// SIMATIC S7-200 project (STEP 7-Micro/WIN), CPU 224 REL 01.22

SYMBOL_TABLE USR1
SAB3             I0.0     //  油泵电机启动
SAB4             I0.1     // 油泵电机停止
SAB5，6           I0.2     // 主轴正转
SAB7，8，9         I0.3     // 主轴停止
SAB10，11         I0.4     // 主轴反转
SAB12，13，14      I0.5     // 主轴正点动
SAB15，16，17      I0.6     // 主轴反点动
SP1，2，FR1        I0.7     // 油压正常
SL1              I1.0     // 回油泵启动
SL2              I1.1     // 回油泵制动
SQ3，SQ4          I1.2     // 主轴变档到位
SQ3，SQ5          I1.3     // 主轴变档到位
SQ3，SQ6          I1.4     // 主轴变档到位
SQ3，SQ7          I1.5     // 主轴变档到位
SP3              I2.0     // 过滤器堵塞
SP4              I2.1     // 过滤器堵塞
KAL1             I2.2     // 驱动器零速输出
KAL2             I2.3     // 驱动器正常输出
KAL3             I2.4     // 驱动器准备输出
SAB18            I2.5     // 套筒电机前进
SAB20            I2.6     // 套筒电机后退
SAB22            I2.7     // 尾座电机前进
SAB24            I3.0     // 尾座电机后退
SAB26            I3.1     // 左溜板箱油泵电机启动
SAB27            I3.2     // 左溜板箱油泵电机停止
SAB28            I3.3     // 左刀架油泵启动
SAB29            I3.4     // 移动停止
SAB30            I3.5     // 正转（前进）
SAB31            I3.6     // 反转（后退）
FR5              I3.7     // 溜板油泵保护
FR6              I4.0     // 刀架油泵保护
SQ8              I4.1     // 左刀架前进限位
SA3              I4.2     // 工作制选择-------给进
SA3，             I4.3     // 工作制选择-------快速
ZYZY             I4.5     // 左刀架1档---------左右
ZYQH             I4.4     // 左刀架1档---------前后
ZEZY             I4.7     // 左刀架2档---------左右
ZEQH             I4.6     // 左刀架2档---------前后
SQ9              I5.0     // 右刀架后退限位
SAB32            I5.1     // 右刀架溜板箱油泵电机启动
SAB33            I5.2     // 右刀架溜板箱油泵电机停止
SAB34            I5.3     // 右刀架油泵启动
SAB35            I5.4     // 右刀架移动停止
SAB36            I5.5     // 右刀架正转（前进）
SAB37            I5.6     // 右刀架反转（后退）
FR7              I5.7     // 右刀架溜板油泵保护
FR8              I6.0     // 刀架油泵保护
SQ10             I6.1     // 两刀架防相撞限位
SA6              I6.3     // 工作制选择----------给进
SA61             I6.2     // 工作制选择----------快速
YYZY             I6.6     // 右刀架1档---------左右
YYQH             I6.7     // 右刀架1档---------前后
YEZY             I6.4     // 右刀架2档---------左右
YEQH             I6.5     // 右刀架2档---------前进
KA0              I7.0     // 急停信号
SA5Y             I7.1     // 主轴变档--------1档
SA5E             I7.2     // 主轴变档--------2档
SA5S             I7.3     // 主轴变档--------3档
DYMKZBH          I7.4     // 驱动器信号
FR611            I7.5     // 驱动器过热信号
KSKZ611          I7.6     // 驱动器开始控制信号
SAB38，39         I7.7     // 主轴升速
SAB40，41         I8.0     // 主轴降速
SAB44，45         I8.7
KA1              Q0.0     // 油泵电机
KA2              Q0.1     // 辅助电源
KA3              Q0.2     // 油泵正常
KA4              Q0.3     // 主电机使能
KA5              Q0.4     // 主电机点动
KA6              Q0.5     // 主电机启动
KA7              Q0.6     // 油压报警
KA8              Q0.7     // 主轴变档电磁阀
KA9              Q1.0     // 主轴变档电磁阀
KA10             Q1.1     // 主轴变档电磁阀
KA11             Q2.0     // 主轴变档电磁阀
KA12             Q2.1     // 主轴1指示
KA13             Q2.2     // 主轴2指示
KA14             Q2.3     // 主轴3指示
HL12             Q2.4     // 过滤器清洗指示
HL13             Q2.5     // 过滤器清洗指示
KA15             Q2.6     // 套筒正转
KA16             Q2.7     // 套筒反转
KA17             Q3.0     // 尾座正转
KA18             Q3.1     // 尾座反转
HL14             Q3.2     // 快速移动指示
HL15             Q3.3     // 进给移动指示
HL16             Q3.4     // 左刀架-----横向移动1
HL17             Q3.5     // 左刀架-----横向移动2
HL18             Q3.6     // 左刀架-----纵向移动1
HL19             Q3.7     // 左刀架-----纵向移动2
KA19             Q4.0     // 左刀架变速传动-------1档
KA20             Q4.1     // 左刀架变速传动-------2档
KA21             Q4.2     // 左刀架变速纵向传动
KA22             Q4.3     // 左刀架变速横向传动
KA23             Q4.4     // 左刀架纵向制动
KA24             Q4.5     // 左刀架横向制动
KA25             Q4.6     // 左溜板油泵
KA26             Q4.7     // 左刀架油泵
KA27             Q5.0     // 回油泵（备用）
KA28             Q5.1
HL20             Q5.2     // 左刀架快速移动指示
HL21             Q5.3     // 左刀架给进移动指示
HL22             Q5.4     // 左刀架横向移动1
HL23             Q5.5     // 左刀架横向移动2
HL24             Q5.6     // 左刀架纵向移动1
HL25             Q5.7     // 左刀架纵向移动2
KA29             Q6.0     // 右刀架变速传动1档
KA30             Q6.1     // 右刀架变速传动2档
KA31             Q6.2     // 右刀架变速纵向传动
KA32             Q6.3     // 右刀架变速横向传动
KA33             Q6.4     // 右刀架变速纵向制动
KA34             Q6.5     // 右刀架变速横向制动
KA35             Q6.6     // 右溜板油泵
KA36             Q6.7     // 右刀架油泵
KA37             Q7.0     // 脉冲使能信号
KA38             Q7.1     // 控制使能信号
KA39             Q7.2     // 内部接触器控制
KA40             Q7.3     // 脉冲使能信号
KA41             Q7.4     // 控制使能信号
KA42             Q7.5     // 控制使能信号
KA43             Q7.6     // 选择电流控制方式
KA44             Q7.7     // 选择电流控制方式
KA45             Q8.1
KA46             Q8.2
KAJT             Q8.7
ZDJZZ            M1.0     // 左刀架正转标志位
ZDJFZ            M1.1     // 左刀架反转标志位
YDJZZ            M1.2     // 右刀架正转标志位
YDJFZ            M1.3     // 右刀架反转标志位
                 M5.2     // 主轴正转标志位
                 M5.3     // 主轴反转标志位
END_SYMBOL_TABLE

ORGANIZATION_BLOCK MAIN:OB1
TITLE=我设计了一个机床润滑系统的核心部件的程序。代码比较复杂，不知道具体实地应用如何，我写一下程序的实现目标以供参考。代码最后更新于2005年2月17号
// 实现目标：操作员通过主轴正转按钮、主轴反转按钮、主轴正点动按钮和主轴反点动按钮控制主轴方向，主电机启动信号驱动主轴连续旋转，主电机点动信号用于短暂调整。主轴模拟输出根据主轴升速按钮和主轴降速按钮调节转速。主轴1档选择开关、主轴2档选择开关和主轴3档选择开关分别触发主轴变档电磁阀1、主轴变档电磁阀2等，档位到位由主轴变档1到位传感器等确认，主轴1档指示灯等显示当前状态。
// 左刀架和右刀架可独立运行。左刀架正转按钮和左刀架反转按钮控制左刀架移动，右刀架正转按钮和右刀架反转按钮控制右刀架移动。左刀架给进模式开关和右刀架给进模式开关选择低速精确加工并调节左刀架模拟输出和右刀架模拟输出，左刀架快速模式开关和右刀架快速模式开关选择高速移动并调整相应输出。左刀架前进限位传感器和右刀架后退限位传感器防止超行程，左刀架防撞限位传感器检测两刀架距离。左刀架正转标志和右刀架反转标志的控制需注意避免相向移动导致碰撞，操作员应谨慎操作。
// 过滤器堵塞传感器1和过滤器堵塞传感器2检测到堵塞时，过滤器清洗指示灯1和过滤器清洗指示灯2亮起，提示维护。套筒电机前进按钮和套筒电机后退按钮分别驱动套筒正转信号和套筒反转信号。尾座电机前进按钮和尾座电机后退按钮分别驱动尾座正转信号和尾座反转信号。
// 紧急停止信号置位后，提示操作员机床处于停止状态。紧急停止按钮被按下时，紧急停止信号置位，操作员需手动复位油泵电机输出、主电机启动信号、套筒正转信号、尾座正转信号、主轴模拟输出、左刀架模拟输出和右刀架模拟输出，确保机床安全。
// 
BEGIN
Network 1
// 611驱动器准备
LD     SM0.0
CALL   SIEMENS611:SBR0
?000
Network 2
// 左刀架运行
LD     SM0.0
CALL   ZDJYX:SBR2
Network 3
// 右刀架运行
LD     SM0.0
CALL   YDJYX:SBR3
Network 4
// 主轴运行
LD     SM0.0
CALL   ZZYX:SBR1
Network 5
// 主轴模拟信号采样
LD     SM0.0
CALL   ZZMNXHCY:SBR4
Network 6
// 油泵电机启动
LD     SAB3:I0.0
O      KA1:Q0.0
AN     SAB4:I0.1
=      KA1:Q0.0
Network 7
// 过滤器清洗
LD     SP3:I2.0
=      HL12:Q2.4
Network 8
// 过滤器清洗
LD     SP4:I2.1
=      HL13:Q2.5
Network 9
// 套筒电机正转
LD     SAB18:I2.5
AN     SAB20:I2.6
=      KA15:Q2.6
Network 10
// 套筒电机反转
LD     SAB20:I2.6
AN     SAB18:I2.5
=      KA16:Q2.7
Network 11
// 尾座电机正转
LD     SAB22:I2.7
AN     SAB24:I3.0
=      KA17:Q3.0
Network 12
// 尾座电机反转
LD     SAB24:I3.0
AN     SAB22:I2.7
=      KA18:Q3.1
Network 13
// 回油泵工作
LD     SL1:I1.0
O      KA27:Q5.0
AN     SL2:I1.1
=      KA27:Q5.0
Network 14
LD     KA1:Q0.0
AN     SP1，2，FR1:I0.7
AN     T204
TON    T203, +20
Network 15
LD     T203
=      M12.0
TON    T204, +20
Network 16
// 报警
LDN    SP1，2，FR1:I0.7
LD     SAB5，6:I0.2
O      SAB10，11:I0.4
O      SAB12，13，14:I0.5
O      SAB15，16，17:I0.6
ALD
O      M12.0
=      KA7:Q0.6
Network 17
LDN    SAB44，45:I8.7
=      KAJT:Q8.7
END_ORGANIZATION_BLOCK

SUBROUTINE_BLOCK SIEMENS611:SBR0
TITLE=子例行程序注释
BEGIN
Network 1 // 网络标题
// 网络注释
LD     M7.0
AN     T108
=      KA39:Q7.2
TON    T250, +10
Network 2
LD     T250
AN     T107
=      KA37:Q7.0
TON    T101, +10
Network 3
LD     T101
AN     T106
=      KA38:Q7.1
TON    T102, +10
Network 4
LD     T102
AN     T105
LPS
TON    T103, +10
A      SA3:I4.2
=      KA43:Q7.6
LPP
A      SA6:I6.3
=      KA44:Q7.7
Network 5
LD     T103
AN     M7.1
=      KA40:Q7.3
Network 6
LD     M7.1
=      M0.0
TON    T105, +10
TON    T106, +20
TON    T107, +30
TON    T108, +40
Network 7
LD     SAB26:I3.1
O      SAB32:I5.1
LD     T109
NOT
A      M7.0
OLD
=      M7.0
Network 8
LD     M7.2
A      M7.3
LD     SAB26:I3.1
O      SAB32:I5.1
NOT
A      M7.1
OLD
=      M7.1
Network 9
LD     M7.1
=      M7.4
TON    T109, +45
Network 10
LD     SAB27:I3.2
LD     SAB26:I3.1
O      SAB32:I5.1
NOT
A      M7.2
OLD
=      M7.2
Network 11
LD     SAB33:I5.2
LD     SAB32:I5.1
O      SAB26:I3.1
NOT
A      M7.3
OLD
=      M7.3
END_SUBROUTINE_BLOCK

SUBROUTINE_BLOCK ZZYX:SBR1
TITLE=子例行程序注释
BEGIN
Network 1
// 辅助电源
LD     KA1:Q0.0
A      SP1，2，FR1:I0.7
=      KA2:Q0.1
TON    T37, +20
Network 2
// 停车信号
LD     T37
=      KA3:Q0.2
TON    T38, +20
Network 3
// 给启动信号
LD     T38
=      KA4:Q0.3
Network 4
// 正转标志位
LD     SAB5，6:I0.2
O      M5.2
LD     SAB7，8，9:I0.3
O      KA41:Q7.4
O      KA42:Q7.5
ALD
AN     SAB10，11:I0.4
AN     SAB15，16，17:I0.6
AN     SAB12，13，14:I0.5
A      KAL2:I2.3
=      M5.2
Network 5
// 反转标志位
LD     SAB10，11:I0.4
O      M5.3
LD     SAB7，8，9:I0.3
O      KA41:Q7.4
O      KA42:Q7.5
ALD
AN     SAB5，6:I0.2
AN     SAB15，16，17:I0.6
AN     SAB12，13，14:I0.5
A      KAL2:I2.3
=      M5.3
Network 6
// 主轴连动
LD     M5.2
O      M5.3
O      M24.0
O      M24.1
O      M25.0
O      M25.1
O      M25.2
A      SP1，2，FR1:I0.7
=      KA6:Q0.5
Network 7
LD     SAB12，13，14:I0.5
AN     SAB15，16，17:I0.6
=      M24.0
Network 8
LD     SAB15，16，17:I0.6
AN     SAB12，13，14:I0.5
=      M24.1
Network 9
LD     M24.0
O      M24.1
=      KA5:Q0.4
Network 10 // 网络标题
// 主轴变挡到位
LD     SQ3，SQ4:I1.2
=      M3.0
Network 11
// 主轴变挡到位
LD     SQ3，SQ5:I1.3
=      M3.1
Network 12
// 主轴变挡到位
LD     SQ3，SQ6:I1.4
=      M3.2
Network 13
// 主轴变挡到位
LD     SQ3，SQ7:I1.5
=      M3.3
Network 14
// 主轴1档
LD     SA5Y:I7.1
LDN    KAL1:I2.2
A      M3.4
OLD
AN     M3.6
AN     M4.0
=      M3.4
=      M3.5
Network 15
// 主轴1档指示灯
LD     M3.5
A      M3.1
A      M3.2
=      KA12:Q2.1
Network 16
// 主轴2档
LD     SA5E:I7.2
LDN    KAL1:I2.2
A      M3.6
OLD
AN     M3.4
AN     M4.0
=      M3.6
=      M3.7
Network 17
// 主轴2档指示灯
LD     M3.7
A      M3.0
A      M3.2
=      KA13:Q2.2
Network 18
// 主轴3档
LD     SA5S:I7.3
LDN    KAL1:I2.2
A      M4.0
OLD
AN     M3.4
AN     M3.6
=      M4.0
=      M4.1
Network 19
// 主轴3档指示灯
LD     M4.1
A      M3.1
A      M3.3
=      KA14:Q2.3
Network 20
// 电磁阀1
LD     M3.7
=      KA8:Q0.7
Network 21
// 电磁阀2
LD     M4.1
O      M3.5
=      KA9:Q1.0
Network 22
// 电磁阀3
LD     M3.5
O      M3.7
=      KA10:Q1.1
Network 23
// 电磁阀4
LD     M4.1
=      KA11:Q2.0
Network 24
// 1档换档脉动
LD     SA5Y:I7.1
LDN    M3.1
ON     M3.2
ALD
AN     T253
TON    T34, +800
Network 25
LDN    T34
TON    T253, +40
=      M25.0
Network 26
// 2档换档脉动
LD     SA5E:I7.2
LDN    M3.0
ON     M3.2
ALD
AN     T254
TON    T35, +200
Network 27
LD     T35
TON    T254, +40
=      M25.1
Network 28
// 3档换档脉动
LD     SA5S:I7.3
LDN    M3.1
ON     M3.3
ALD
AN     T255
TON    T36, +200
Network 29
LD     T36
TON    T255, +40
=      M25.2
END_SUBROUTINE_BLOCK

SUBROUTINE_BLOCK ZDJYX:SBR2
TITLE=子例行程序注释
BEGIN
Network 1
// 给定快速和给定速度范围
LD     SM0.0
LPS
A      SA3，:I4.3
LPS
A      M20.0
MOVW   +25000, AQW4
LPP
A      M20.1
MOVW   -25000, AQW4
LPP
A      SA3:I4.2
LPS
AW<=   AIW2, +32000
MOVW   AIW2, VW20
LPP
AW>=   AIW2, +32000
MOVW   +32000, VW20
Network 2
LD     SA3:I4.2
A      ZDJZZ:M1.0
AN     ZDJFZ:M1.1
MOVW   VW20, VW21
Network 3
// 选择速度范围
LD     SA3:I4.2
A      ZDJZZ:M1.0
AN     ZDJFZ:M1.1
AW<=   VW21, +32000
AW>=   VW21, +0
MOVW   VW21, AQW4
Network 4
// 改变方向
LD     SA3:I4.2
A      ZDJFZ:M1.1
AN     ZDJZZ:M1.0
MOVW   -1, VW200
*I     VW20, VW200
Network 5
LD     SA3:I4.2
A      ZDJFZ:M1.1
AN     ZDJZZ:M1.0
MOVW   VW200, VW201
Network 6
// 选择速度范围
LD     SA3:I4.2
A      ZDJFZ:M1.1
AN     ZDJZZ:M1.0
AW<=   VW201, +0
AW>=   VW201, -32000
MOVW   VW201, AQW4
Network 7
// 左溜板箱油泵电机
LD     SAB26:I3.1
O      KA25:Q4.6
AN     SAB27:I3.2
AN     FR5:I3.7
=      KA25:Q4.6
TON    T111, +3000
Network 8
// 左刀架油泵电机
LD     KA25:Q4.6
LD     SA3，:I4.3
LD     M20.0
O      M20.1
ALD
OLD
LDN    T111
O      M1.6
ALD
AN     FR6:I4.0
=      KA26:Q4.7
Network 9
// 左刀架油泵启动
LD     SAB28:I3.3
O      M1.6
AN     T112
=      M1.6
TON    T112, +3000
Network 10
// 左刀架工作方式选择
LD     KA25:Q4.6
LPS
AN     KAL1:I2.2
LD     SA3:I4.2
O      KA41:Q7.4
ALD
AN     HL14:Q3.2
=      HL15:Q3.3
LPP
A      SA3，:I4.3
AN     HL15:Q3.3
=      HL14:Q3.2
Network 11
// 左刀架1档左右
LD     KA25:Q4.6
LD     ZYZY:I4.5
O      KA41:Q7.4
ALD
AN     M2.0
AN     M2.1
AN     M2.2
=      HL16:Q3.4
=      M1.7
Network 12
// 左刀架1档前后
LD     KA25:Q4.6
LD     ZYQH:I4.4
O      KA41:Q7.4
ALD
AN     M1.7
AN     M2.1
AN     M2.2
=      HL18:Q3.6
=      M2.0
Network 13
// 左刀架2档左右
LD     KA25:Q4.6
LD     ZEZY:I4.7
O      KA41:Q7.4
ALD
AN     M1.7
AN     M2.0
AN     M2.2
=      HL17:Q3.5
=      M2.1
Network 14
// 左刀架2档前后
LD     KA25:Q4.6
LD     ZEQH:I4.6
O      KA41:Q7.4
ALD
AN     M1.7
AN     M2.0
AN     M2.1
=      HL19:Q3.7
=      M2.2
Network 15
// 左刀架电机正转
LD     SAB30:I3.5
O      ZDJZZ:M1.0
AN     SAB29:I3.4
A      SA3:I4.2
AN     ZDJFZ:M1.1
A      SQ8:I4.1
A      SP1，2，FR1:I0.7
AN     KAL1:I2.2
=      ZDJZZ:M1.0
Network 16
// 左刀架电机正点动
LD     SA3，:I4.3
AN     SA3:I4.2
A      SAB30:I3.5
AN     ZDJFZ:M1.1
=      M20.0
Network 17
// 左刀架电机反转
LD     SAB31:I3.6
O      ZDJFZ:M1.1
AN     SAB29:I3.4
A      SA3:I4.2
AN     ZDJZZ:M1.0
AN     SQ10:I6.1
A      SP1，2，FR1:I0.7
AN     KAL1:I2.2
=      ZDJFZ:M1.1
Network 18
// 左刀架电机反点动
LD     SA3，:I4.3
AN     SA3:I4.2
A      SAB31:I3.6
AN     ZDJZZ:M1.0
=      M20.1
Network 19
// 给定611启动信号
LD     ZDJZZ:M1.0
O      ZDJFZ:M1.1
AW>=   AIW2, +45
LD     M20.0
O      M20.1
OLD
=      KA41:Q7.4
Network 20
// 左刀架变速传动-------1档电磁阀
LD     M1.7
O      M2.0
A      SA3:I4.2
=      KA19:Q4.0
Network 21
// 给进状态下左刀架变速传动-------2档电磁阀标志位
LD     M2.1
O      M2.2
A      SA3:I4.2
=      M20.2
Network 22
// 快速状态下左刀架变速传动-------2档电磁阀标志位
LD     M2.1
O      M2.2
O      M1.7
O      M2.0
A      SA3，:I4.3
=      M20.3
Network 23
// 左刀架变速传动-------2档电磁阀
LD     M20.2
O      M20.3
=      KA20:Q4.1
Network 24
// 左刀架变速纵向传动电磁阀
LD     M2.0
O      M2.2
=      KA21:Q4.2
Network 25
// 左刀架变速横向传动电磁阀
LD     M1.7
O      M2.1
=      KA22:Q4.3
Network 26
// 左刀架纵向制动电磁阀
LD     M1.7
O      M2.1
LD     ZDJZZ:M1.0
O      ZDJFZ:M1.1
ALD
=      KA23:Q4.4
Network 27
// 左刀架横向制动电磁阀
LD     M2.0
O      M2.2
LD     ZDJZZ:M1.0
O      ZDJFZ:M1.1
ALD
=      KA24:Q4.5
END_SUBROUTINE_BLOCK

SUBROUTINE_BLOCK YDJYX:SBR3
TITLE=
BEGIN
Network 1
// 给定快速和给定速度范围
LD     SM0.0
LPS
A      SA61:I6.2
LPS
A      M21.0
MOVW   +25000, AQW6
LPP
A      M21.1
MOVW   -25000, AQW6
LPP
A      SA6:I6.3
LPS
AW<=   AIW4, +32000
MOVW   AIW4, VW40
LPP
AW>=   AIW4, +32000
MOVW   +32000, VW40
Network 2
LD     SA6:I6.3
A      YDJZZ:M1.2
AN     YDJFZ:M1.3
MOVW   VW40, VW41
Network 3
// 选择速度范围
LD     SA6:I6.3
A      YDJZZ:M1.2
AN     YDJFZ:M1.3
AW<=   VW41, +32000
AW>=   VW41, +0
MOVW   VW41, AQW6
Network 4
// 改变方向
LD     SA6:I6.3
A      YDJFZ:M1.3
AN     YDJZZ:M1.2
MOVW   -1, VW400
*I     VW40, VW400
Network 5
LD     SA6:I6.3
A      YDJFZ:M1.3
AN     YDJZZ:M1.2
MOVW   VW400, VW401
Network 6
// 选择速度范围
LD     SA6:I6.3
A      YDJFZ:M1.3
AN     YDJZZ:M1.2
AW<=   VW401, +0
AW>=   VW401, -32000
MOVW   VW401, AQW6
Network 7
// 右溜板箱油泵电机
LD     SAB32:I5.1
O      KA35:Q6.6
AN     SAB33:I5.2
AN     FR7:I5.7
=      KA35:Q6.6
TON    T114, +3000
Network 8
// 右刀架油泵电机
LD     KA35:Q6.6
LD     SA61:I6.2
LD     M21.0
O      M21.1
ALD
OLD
LDN    T114
O      M9.0
ALD
AN     FR8:I6.0
=      KA36:Q6.7
Network 9
// 右刀架油泵启动
LD     SAB34:I5.3
O      M9.0
AN     T115
=      M9.0
TON    T115, +3000
Network 10
// 右刀架工作方式
LD     KA35:Q6.6
LPS
AN     KAL1:I2.2
LD     SA6:I6.3
O      KA42:Q7.5
ALD
AN     HL20:Q5.2
=      HL21:Q5.3
LPP
A      SA61:I6.2
AN     HL21:Q5.3
=      HL20:Q5.2
Network 11
// 右刀架1档左右
LD     KA35:Q6.6
LD     YYZY:I6.6
O      KA42:Q7.5
ALD
AN     M2.3
AN     M2.5
AN     M2.6
=      HL22:Q5.4
=      M2.4
Network 12
// 右刀架1档前后
LD     KA35:Q6.6
LD     YYQH:I6.7
O      KA42:Q7.5
ALD
AN     M2.4
AN     M2.5
AN     M2.6
=      HL24:Q5.6
=      M2.3
Network 13
// 右刀架2档左右
LD     KA35:Q6.6
LD     YEZY:I6.4
O      KA42:Q7.5
ALD
AN     M2.3
AN     M2.4
AN     M2.5
=      HL23:Q5.5
=      M2.6
Network 14
// 右刀架2档前后
LD     KA35:Q6.6
LD     YEQH:I6.5
O      KA42:Q7.5
ALD
AN     M2.3
AN     M2.4
AN     M2.6
=      HL25:Q5.7
=      M2.5
Network 15
// 右刀架电机正转
LD     SAB36:I5.5
O      YDJZZ:M1.2
AN     SAB35:I5.4
A      SA6:I6.3
AN     YDJFZ:M1.3
AN     SQ10:I6.1
A      SP1，2，FR1:I0.7
AN     KAL1:I2.2
=      YDJZZ:M1.2
Network 16
// 右刀架电机正点动
LD     SA61:I6.2
A      SAB36:I5.5
AN     SA6:I6.3
AN     YDJFZ:M1.3
=      M21.0
Network 17
// 右架电机反转
LD     SAB37:I5.6
O      YDJFZ:M1.3
AN     SAB35:I5.4
A      SA6:I6.3
AN     YDJZZ:M1.2
AN     SQ9:I5.0
A      SP1，2，FR1:I0.7
AN     KAL1:I2.2
=      YDJFZ:M1.3
Network 18
// 右架电机反点动
LD     SA61:I6.2
A      SAB37:I5.6
AN     SA6:I6.3
AN     YDJZZ:M1.2
=      M21.1
Network 19
// 给定611启动信号
LD     YDJZZ:M1.2
O      YDJFZ:M1.3
AW>=   AIW4, +40
LD     M21.0
O      M21.1
OLD
=      KA42:Q7.5
Network 20
// 右刀架变速传动-------1档电磁阀
LD     M2.3
O      M2.4
A      SA6:I6.3
=      KA29:Q6.0
Network 21
// 给进状态下右刀架变速传动-------2档电磁阀标志位
LD     M2.5
O      M2.6
A      SA6:I6.3
=      M21.2
Network 22
// 快进状态下右刀架变速传动-------2档电磁阀标志位
LD     M2.3
O      M2.4
O      M2.5
O      M2.6
A      SA61:I6.2
=      M21.3
Network 23
// 右刀架变速传动-------2档电磁阀
LD     M21.2
O      M21.3
=      KA30:Q6.1
Network 24
// 右刀架变速纵向传动电磁阀
LD     M2.3
O      M2.5
=      KA31:Q6.2
Network 25
// 右刀架变速横向传动电磁阀
LD     M2.4
O      M2.6
=      KA32:Q6.3
Network 26
// 右刀架纵向制动电磁阀
LD     M2.4
O      M2.6
LD     YDJZZ:M1.2
O      YDJFZ:M1.3
ALD
=      KA33:Q6.4
Network 27
// 右刀架横向制动电磁阀
LD     M2.3
O      M2.5
LD     YDJZZ:M1.2
O      YDJFZ:M1.3
ALD
=      KA34:Q6.5
END_SUBROUTINE_BLOCK

SUBROUTINE_BLOCK ZZMNXHCY:SBR4
TITLE=子例行程序注释
BEGIN
Network 1
// 1档正转的初始速度
LD     M3.4
A      M5.2
AN     M5.3
AN     SAB12，13，14:I0.5
AN     SAB15，16，17:I0.6
MOVW   +1333, VW70
Network 2
// 1档反转的初始速度
LD     M3.4
A      M5.3
AN     M5.2
AN     SAB12，13，14:I0.5
AN     SAB15，16，17:I0.6
MOVW   -1333, VW71
Network 3
// 正点动给定速度
LD     M24.0
O      M25.0
O      M25.1
O      M25.2
MOVW   +16000, AQW0
Network 4
// 反点动给定速度
LD     M24.1
MOVW   -16000, AQW0
Network 5
// 2/3档正转初始速度
LD     M3.6
O      M4.0
A      M5.2
MOVW   +10666, VW72
Network 6
// 2/3档反转初始速度
LD     M3.6
O      M4.0
A      M5.3
MOVW   -10666, VW73
Network 7
LD     SAB38，39:I7.7
TON    T200, +10
Network 8
LD     T200
AN     T98
TON    T97, +6
Network 9
LD     T97
TON    T98, +6
Network 10
LD     T97
=      M11.0
Network 11
LD     SAB40，41:I8.0
TON    T201, +10
Network 12
LD     T201
AN     T100
TON    T99, +6
Network 13
LD     T99
TON    T100, +6
Network 14
LD     T99
=      M11.1
Network 15
// 1档计数
LD     SAB38，39:I7.7
AN     T200
O      M11.0
AN     SAB40，41:I8.0
A      M3.4
AN     C0
LD     SAB40，41:I8.0
AN     T201
O      M11.1
AN     SAB38，39:I7.7
A      M3.4
AN     M14.0
LD     SM0.1
CTUD   C0, +75
Network 16
LDW<=  C0, +0
=      M14.0
Network 17
// 2/3档计数
LD     SAB38，39:I7.7
AN     T200
O      M11.0
AN     SAB40，41:I8.0
LD     M3.6
O      M4.0
ALD
AN     C1
LD     SAB40，41:I8.0
AN     T201
O      M11.1
AN     SAB38，39:I7.7
LD     M3.6
O      M4.0
ALD
AN     M14.1
LD     SM0.1
CTUD   C1, +53
Network 18
LDW<=  C1, +0
=      M14.1
Network 19
LD     M3.4
A      M5.2
AN     M5.3
MOVW   C0, VW74
*I     +400, VW74
Network 20
LD     M3.4
A      M5.2
AN     M5.3
MOVW   VW70, VW80
+I     VW74, VW80
Network 21
LD     M3.4
A      M5.3
AN     M5.2
MOVW   C0, VW75
*I     -400, VW75
Network 22
LD     M3.4
A      M5.3
AN     M5.2
MOVW   VW71, VW80
+I     VW75, VW80
Network 23
LD     M3.6
O      M4.0
A      M5.2
AN     M5.3
MOVW   C1, VW76
*I     +400, VW76
Network 24
LD     M3.6
O      M4.0
A      M5.2
AN     M5.3
MOVW   VW72, VW81
+I     VW76, VW81
Network 25
LD     M3.6
O      M4.0
A      M5.3
AN     M5.2
MOVW   C1, VW77
*I     -400, VW77
Network 26
LD     M5.3
LD     M3.6
O      M4.0
ALD
AN     M5.2
MOVW   VW73, VW81
+I     VW77, VW81
Network 27
// 1档正转速度选择范围
LD     M3.4
A      M5.2
AN     M5.3
AW<=   VW80, +32000
AW>=   VW80, +1333
MOVW   VW80, AQW0
Network 28
// 1档反转速度选择范围
LD     M3.4
A      M5.3
AN     M5.2
AW<=   VW80, -1333
AW>=   VW80, -32000
MOVW   VW80, AQW0
Network 29
// 2/3档正转速度选择范围
LD     M3.6
O      M4.0
A      M5.2
AN     M5.3
AW<=   VW81, +32000
AW>=   VW81, +10666
MOVW   VW81, AQW0
Network 30
// 2/3档反转速度选择范围
LD     M3.6
O      M4.0
A      M5.3
AN     M5.2
AW<=   VW81, -10666
AW>=   VW81, -32000
MOVW   VW81, AQW0
END_SUBROUTINE_BLOCK
